TYPE EM_Machine_WRN :
STRUCT
END_STRUCT
END_TYPE

(* stored: Version 1.1.0.1, ProductVersion 3.1.4024.12
   DUT EM_Machine_WRN: Id {d68fecdb-7924-4ae0-83e0-6438ee2b481d} *)
